# EPICS autosave request: gardasoftLED/PP420LED_settings.req
$(P):BRIGHTNESS
$(P):PERIOD
